// TwinCAT 3 PLC project ads
// ProgramVersion: 3.1.4022.4
// libraries:
//   Tc2_Standard, * (Beckhoff Automation GmbH)
//   Tc2_System, * (Beckhoff Automation GmbH)
//   Tc3_Module, * (Beckhoff Automation GmbH)
// project tree:
//   DUTs/ ComplexStruct.TcDUT, PLCStruct.TcDUT, SimpleStruct.TcDUT
//   / PlcTask.TcTTO
//   POUs/ MAIN.TcPOU
// real-time tasks:
//   TASK PlcTask: cycle T#10ms, priority 20, ADS port 350

CONFIGURATION ads
    RESOURCE PLC ON TwinCAT3
        TASK PlcTask(INTERVAL := T#10ms, PRIORITY := 20);
        PROGRAM MAIN WITH PlcTask : MAIN;
    END_RESOURCE
END_CONFIGURATION

// ---- DUTs/ComplexStruct.TcDUT
TYPE ComplexStruct :
STRUCT
	intVal	:INT:=100;
	DintArr: ARRAY[1..5] OF DINT := [1, 2, 3, 4,100];
	BoolVal	:BOOL:= TRUE;
	ByteVal	:BYTE:=12;
	LrealVal	:LREAL:= 123.67;
	strVal 	:STRING(10):= 'hello';
	//strArray: ARRAY[1..3] OF STRING(10) := ['abc', 'qwe', 'hjk'];  ??
	SimpleStruct1		:SimpleStruct;	
END_STRUCT
END_TYPE

// ---- DUTs/PLCStruct.TcDUT
TYPE PLCStruct :
STRUCT
	intVal   : INT;  (*Offset 0*) 
  	dintVal  : DINT; (*Offset 2*) 
  	byteVal  : SINT; (*Offset 6*)  
  	lrealVal : LREAL;(*Offset 7*) 
  	realVal  : REAL; (*Offset 15 --> Total size 19 Bytes*) 
END_STRUCT
END_TYPE

// ---- DUTs/SimpleStruct.TcDUT
TYPE SimpleStruct :
STRUCT
	lrealVal	:LREAL:= 1.23;
	dintVal		:DINT:= 120000;
END_STRUCT
END_TYPE

// ---- POUs/MAIN.TcPOU
PROGRAM MAIN
VAR	
// primitiv datatype

	int1 :INT:=100;
	bool1	:BOOL:= TRUE;
	dint1	:DINT:= 101;
	byte1	:BYTE:= 10;
	real1	:REAL:=123.45;
	lreal1	:LREAL:= 56.78;	
	
	str1	:STRING(50):= 'JOT';
	str2	:STRING(50):= 'MAG';
	i:INT;
	intArray: ARRAY [1..10] OF INT := [11, 12, 13, 14, 15, 16, 17, 18, 19, 20];
	DintArray1	: ARRAY[1..10] OF DINT;
	complexStruct		:ComplexStruct;
	
	PLCVar		:PLCStruct;
END_VAR

//Reading and writing PLC variables of anytype
;

END_PROGRAM
